VAR_GLOBAL
	FioInputs : ARRAY [0..15] OF BYTE;
	FioOutputs : ARRAY [0..15] OF BYTE;
END_VAR

(* stored: Version 1.1.0.1
   GVL FIO_Modbus: Id {f0652f86-660b-44a4-8347-b07934b026dd} *)
